KUKA KRL program: DAI_CHECK_GRH_01.src, DAI_CHECK_GRH_01.dat

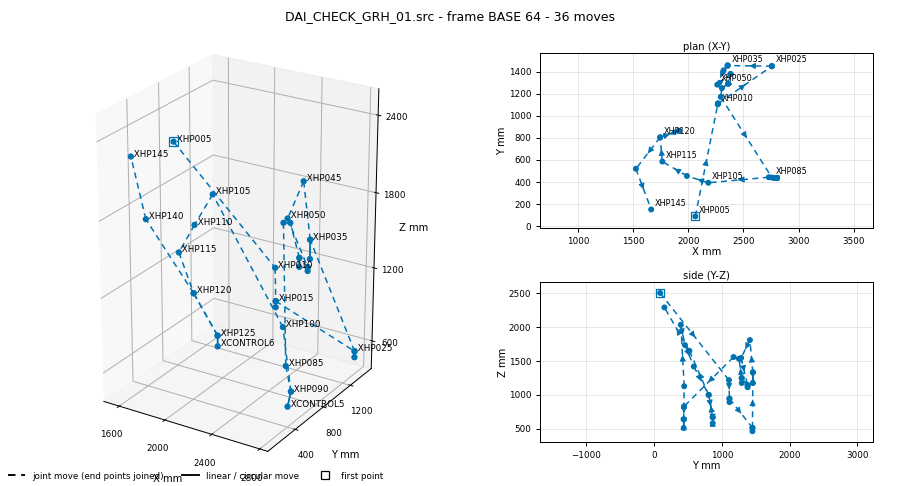
[picture p0: tool path of DAI_CHECK_GRH_01.src in frame BASE 64, 36 of 38 moves have a stored position in this frame; points joined in program order, loops and branches not executed]
--- DAI_CHECK_GRH_01.src ---
&ACCESS RVO
&REL 41
&COMMENT Greiferpruefung
&PARAM TEMPLATE = C:\KRC\roboter\template\vg_appl
&PARAM DISKPATH = KRC:\R1\H_Prog
DEF DAI_CHECK_GRH_01( )
;FOLD INI;%{PE}
  ;FOLD BASISTECH INI
    GLOBAL INTERRUPT DECL 3 WHEN $STOPMESS==TRUE DO IR_STOPM ( )
    INTERRUPT ON 3
    BAS (#INITMOV,0 )
  ;ENDFOLD (BASISTECH INI)
  ;FOLD USER INI
    ;Make your modifications here
  ;ENDFOLD (USER INI)
;ENDFOLD (INI)
;FOLD ; Anlagenbezeichn: HC53_C    Stations-Nr: 060RB_100;%{PE}
;FOLD Parameters ;%{h}
;Params IlfProvider=kukaroboter.basistech.inlineforms.comments.comment; Kuka.Content=Anlagenbezeichn: HC53_C    Stations-Nr: 060RB_100
;ENDFOLD
;ENDFOLD
;FOLD ; Stand / Version: V1.0;%{PE}
;FOLD Parameters ;%{h}
;Params IlfProvider=kukaroboter.basistech.inlineforms.comments.comment; Kuka.Content=Stand / Version: V1.0
;ENDFOLD
;ENDFOLD
;FOLD ; Name Bearbeiter: EBZ-AE;%{PE}
;FOLD Parameters ;%{h}
;Params IlfProvider=kukaroboter.basistech.inlineforms.comments.comment; Kuka.Content=Name Bearbeiter: EBZ-AE
;ENDFOLD
;ENDFOLD
;FOLD ; Translator Version:29.01.2024 - Version 15.08;%{PE}
;FOLD Parameters ;%{h}
;Params IlfProvider=kukaroboter.basistech.inlineforms.comments.comment; Kuka.Content=Translator Version:29.01.2024 - Version 15.08
;ENDFOLD
;ENDFOLD

REPEAT
;FOLD MSG_T1
MSG_SHOW("DAI_H_Prog",#quit,999,"dai_tool_ok_1")
;ENDFOLD

; ***************************************
; A C H T U N G !!! Nur in $T1 abfahren
; ***************************************
UNTIL $T1 == TRUE
;FOLD robot_ok-program
MSG_SHOW("DAI_H_Prog",#quit,999,"dai_rob_ok_0")
DAI_ROBOT_OK ( )
;ENDFOLD

; ***************************************
; Bei Werkzeugwechsel Abfrage ob richtiges Werkzeug angekoppelt ist
; ***************************************
;FOLD MSG_Tool_chg
MSG_BTN("OK")
MSG_SHOW("DAI_H_Prog",#dialog,999,"dai_tool_ok_1",handle,answer)
;ENDFOLD


;FOLD ; This program has been cleaned by KANERT_Makro. High risk of crash!!! Check the program carefully before deleting this comment. ;%{PE}
;FOLD Parameters ;%{h}
;Params IlfProvider=kukaroboter.basistech.inlineforms.comments.comment; Kuka.Content=This program has been cleaned by KANERT_Makro. High risk of crash!!! Check the program carefully before deleting this comment.
;ENDFOLD
WAIT FOR FALSE
;ENDFOLD
;FOLD PTP HOME Vel=100 % DEFAULT;%{PE}
;FOLD Parameters ;%{h}
;Params IlfProvider=kukaroboter.basistech.inlineforms.movement.old; Kuka.IsGlobalPoint=False; Kuka.PointName=HOME; Kuka.BlendingEnabled=False; Kuka.MoveDataPtpName=DEFAULT; Kuka.VelocityPtp=100; Kuka.CurrentCDSetIndex=0; Kuka.MovementParameterFieldEnabled=True; IlfCommand=PTP
;ENDFOLD
$BWDSTART = FALSE
PDAT_ACT = PDEFAULT
FDAT_ACT = FHOME
BAS(#PTP_PARAMS, 100.0)
SET_CD_PARAMS (0)
PTP XHOME
;ENDFOLD

;Dynamische Pruefung Teil vorhanden
;FOLD PartPresent.CheckOff #1:5277, #2:5278, #3:1025, #4:1025, #5:1025, #6:1025, Bounce Time:100, Constant: Yes;%{PE}%
CheckPartPresent(5277,5278,1025,1025,1025,1025,100, True,FALSE)
;ENDFOLD

;Greifer-Ventile betatigen/pruefen
;FOLD DAI_GripValveCheck.Valve2 State:Fixierstift Ausfahren Gs, 060GRH101-QM1;%{PE}%
CheckValveState(2,1)
;ENDFOLD
;FOLD DAI_GripValveCheck.Valve3 State:Spanner Oeffnen Gs, 060GRH101-QM2;%{PE}%
CheckValveState(3,1)
;ENDFOLD
;FOLD DAI_GripValveCheck.Valve4 State:Spanner Oeffnen Gs, 060GRH101-QM3;%{PE}%
CheckValveState(4,1)
;ENDFOLD

;FOLD PTP HP005 Vel=100 % PDAT1 Tool[64]:Zero Base[64]:Zero;%{PE}
;FOLD Parameters ;%{h}
;Params IlfProvider=kukaroboter.basistech.inlineforms.movement.old; Kuka.IsGlobalPoint=False; Kuka.PointName=HP005; Kuka.BlendingEnabled=False; Kuka.MoveDataPtpName=PDAT1; Kuka.VelocityPtp=100; Kuka.CurrentCDSetIndex=0; Kuka.MovementParameterFieldEnabled=True; IlfCommand=PTP
;ENDFOLD
$BWDSTART = FALSE
PDAT_ACT = PPDAT1
FDAT_ACT = FHP005
BAS(#PTP_PARAMS, 100.0)
SET_CD_PARAMS (0)
PTP XHP005
;ENDFOLD
;FOLD PTP HP010 Vel=100 % PDAT2 Tool[64]:Zero Base[64]:Zero;%{PE}
;FOLD Parameters ;%{h}
;Params IlfProvider=kukaroboter.basistech.inlineforms.movement.old; Kuka.IsGlobalPoint=False; Kuka.PointName=HP010; Kuka.BlendingEnabled=False; Kuka.MoveDataPtpName=PDAT2; Kuka.VelocityPtp=100; Kuka.CurrentCDSetIndex=0; Kuka.MovementParameterFieldEnabled=True; IlfCommand=PTP
;ENDFOLD
$BWDSTART = FALSE
PDAT_ACT = PPDAT2
FDAT_ACT = FHP010
BAS(#PTP_PARAMS, 100.0)
SET_CD_PARAMS (0)
PTP XHP010
;ENDFOLD
;FOLD PTP HP015 Vel=100 % PDAT3 Tool[64]:Zero Base[64]:Zero;%{PE}
;FOLD Parameters ;%{h}
;Params IlfProvider=kukaroboter.basistech.inlineforms.movement.old; Kuka.IsGlobalPoint=False; Kuka.PointName=HP015; Kuka.BlendingEnabled=False; Kuka.MoveDataPtpName=PDAT3; Kuka.VelocityPtp=100; Kuka.CurrentCDSetIndex=0; Kuka.MovementParameterFieldEnabled=True; IlfCommand=PTP
;ENDFOLD
$BWDSTART = FALSE
PDAT_ACT = PPDAT3
FDAT_ACT = FHP015
BAS(#PTP_PARAMS, 100.0)
SET_CD_PARAMS (0)
PTP XHP015
;ENDFOLD

; ***************************************
; Stift ausfahren
; ***************************************

; ***************************************
;FOLD Kontrollspitzen anbringen
MSG_BTN("OK")
MSG_SHOW("DAI_H_PROG",#dialog,999,"dai_tool_ok_7",handle,answer)
;ENDFOLD
;FOLD WAIT FOR ( IN 1026 'Vordefinierte Eingang immer ruckgesetzt.' )  ;%{PE}
;FOLD Parameters ;%{h}
;Params IlfProvider=kukaroboter.basistech.inlineforms.logics.waitfor; Kuka.WaitLogicTerm1=None; Kuka.WaitForNot1=False; Kuka.WaitLogicOp2.Term1=None; Kuka.WaitForNot2.Term1=False; Kuka.WaitForSysVar2.Term1=IN; Kuka.WaitForIndex2.Term1=1026; Kuka.WaitForIndexName2.Term1=Vordefinierte Eingang immer ruckgesetzt.; Kuka.WaitForTermNumbers=1; Kuka.WaitForOpNumbers=2; Kuka.WaitForCont=False
;ENDFOLD
WAIT FOR  ( $IN[1026] )
;ENDFOLD

; ***************************************
;FOLD ;Kontrollposition 1 QMXMMYY mit Tool 64 ;%{PE}
;FOLD Parameters ;%{h}
;Params IlfProvider=kukaroboter.basistech.inlineforms.comments.comment; Kuka.Content=Kontrollposition 1 QMXMMYY mit Tool 64
;ENDFOLD
;ENDFOLD
;FOLD LIN CONTROL1 Vel=0.2 m/s CPDAT4 Tool[64]:Zero Base[64]:Zero ;%{PE}
;FOLD Parameters ;%{h}
;Params IlfProvider=kukaroboter.basistech.inlineforms.movement.old; Kuka.IsGlobalPoint=False; Kuka.PointName=CONTROL1; Kuka.BlendingEnabled=False; Kuka.MoveDataName=CPDAT4; Kuka.VelocityPath=0.2; Kuka.CurrentCDSetIndex=0; Kuka.MovementParameterFieldEnabled=True; IlfCommand=LIN
;ENDFOLD
$BWDSTART = FALSE
LDAT_ACT = LCPDAT4
FDAT_ACT = FCONTROL1
BAS(#CP_PARAMS, 0.2)
SET_CD_PARAMS (0)
LIN XCONTROL1
;ENDFOLD

;FOLD WAIT FOR ( IN 1026 'Vordefinierte Eingang immer ruckgesetzt.' )  ;%{PE}
;FOLD Parameters ;%{h}
;Params IlfProvider=kukaroboter.basistech.inlineforms.logics.waitfor; Kuka.WaitLogicTerm1=None; Kuka.WaitForNot1=False; Kuka.WaitLogicOp2.Term1=None; Kuka.WaitForNot2.Term1=False; Kuka.WaitForSysVar2.Term1=IN; Kuka.WaitForIndex2.Term1=1026; Kuka.WaitForIndexName2.Term1=Vordefinierte Eingang immer ruckgesetzt.; Kuka.WaitForTermNumbers=1; Kuka.WaitForOpNumbers=2; Kuka.WaitForCont=False
;ENDFOLD
WAIT FOR  ( $IN[1026] )
;ENDFOLD

;FOLD LIN HP020 Vel=0.2 m/s CPDAT5 Tool[64]:Zero Base[64]:Zero ;%{PE}
;FOLD Parameters ;%{h}
;Params IlfProvider=kukaroboter.basistech.inlineforms.movement.old; Kuka.IsGlobalPoint=False; Kuka.PointName=HP020; Kuka.BlendingEnabled=False; Kuka.MoveDataName=CPDAT5; Kuka.VelocityPath=0.2; Kuka.CurrentCDSetIndex=0; Kuka.MovementParameterFieldEnabled=True; IlfCommand=LIN
;ENDFOLD
$BWDSTART = FALSE
LDAT_ACT = LCPDAT5
FDAT_ACT = FHP020
BAS(#CP_PARAMS, 0.2)
SET_CD_PARAMS (0)
LIN XHP020
;ENDFOLD

; ***************************************
; Die naechsten 3 Punkte werden mit Tool[10] angefahren
; ***************************************
;FOLD PTP HP025 Vel=100 % PDAT6 Tool[10]:GRH_01_ZBHC_O Base[64]:Zero;%{PE}
;FOLD Parameters ;%{h}
;Params IlfProvider=kukaroboter.basistech.inlineforms.movement.old; Kuka.IsGlobalPoint=False; Kuka.PointName=HP025; Kuka.BlendingEnabled=False; Kuka.MoveDataPtpName=PDAT6; Kuka.VelocityPtp=100; Kuka.CurrentCDSetIndex=0; Kuka.MovementParameterFieldEnabled=True; IlfCommand=PTP
;ENDFOLD
$BWDSTART = FALSE
PDAT_ACT = PPDAT6
FDAT_ACT = FHP025
BAS(#PTP_PARAMS, 100.0)
SET_CD_PARAMS (0)
PTP XHP025
;ENDFOLD

;FOLD ; Kontrollposition 1A QM1MM01 mit Tool 10 ;%{PE}
;FOLD Parameters ;%{h}
;Params IlfProvider=kukaroboter.basistech.inlineforms.comments.comment; Kuka.Content=Kontrollposition 1A QM1MM01 mit Tool 10
;ENDFOLD
;ENDFOLD
;FOLD LIN CONTROL1A Vel=0.2 m/s CPDAT7 Tool[10]:GRH_01_ZBHC_O Base[64]:Zero ;%{PE}
;FOLD Parameters ;%{h}
;Params IlfProvider=kukaroboter.basistech.inlineforms.movement.old; Kuka.IsGlobalPoint=False; Kuka.PointName=CONTROL1A; Kuka.BlendingEnabled=False; Kuka.MoveDataName=CPDAT7; Kuka.VelocityPath=0.2; Kuka.CurrentCDSetIndex=0; Kuka.MovementParameterFieldEnabled=True; IlfCommand=LIN
;ENDFOLD
$BWDSTART = FALSE
LDAT_ACT = LCPDAT7
FDAT_ACT = FCONTROL1A
BAS(#CP_PARAMS, 0.2)
SET_CD_PARAMS (0)
LIN XCONTROL1A
;ENDFOLD

;FOLD WAIT FOR ( IN 1026 'Vordefinierte Eingang immer ruckgesetzt.' )  ;%{PE}
;FOLD Parameters ;%{h}
;Params IlfProvider=kukaroboter.basistech.inlineforms.logics.waitfor; Kuka.WaitLogicTerm1=None; Kuka.WaitForNot1=False; Kuka.WaitLogicOp2.Term1=None; Kuka.WaitForNot2.Term1=False; Kuka.WaitForSysVar2.Term1=IN; Kuka.WaitForIndex2.Term1=1026; Kuka.WaitForIndexName2.Term1=Vordefinierte Eingang immer ruckgesetzt.; Kuka.WaitForTermNumbers=1; Kuka.WaitForOpNumbers=2; Kuka.WaitForCont=False
;ENDFOLD
WAIT FOR  ( $IN[1026] )
;ENDFOLD

;FOLD LIN HP030 Vel=0.2 m/s CPDAT8 Tool[10]:GRH_01_ZBHC_O Base[64]:Zero ;%{PE}
;FOLD Parameters ;%{h}
;Params IlfProvider=kukaroboter.basistech.inlineforms.movement.old; Kuka.IsGlobalPoint=False; Kuka.PointName=HP030; Kuka.BlendingEnabled=False; Kuka.MoveDataName=CPDAT8; Kuka.VelocityPath=0.2; Kuka.CurrentCDSetIndex=0; Kuka.MovementParameterFieldEnabled=True; IlfCommand=LIN
;ENDFOLD
$BWDSTART = FALSE
LDAT_ACT = LCPDAT8
FDAT_ACT = FHP030
BAS(#CP_PARAMS, 0.2)
SET_CD_PARAMS (0)
LIN XHP030
;ENDFOLD
;FOLD PTP HP035 Vel=100 % PDAT9 Tool[64]:Zero Base[64]:Zero;%{PE}
;FOLD Parameters ;%{h}
;Params IlfProvider=kukaroboter.basistech.inlineforms.movement.old; Kuka.IsGlobalPoint=False; Kuka.PointName=HP035; Kuka.BlendingEnabled=False; Kuka.MoveDataPtpName=PDAT9; Kuka.VelocityPtp=100; Kuka.CurrentCDSetIndex=0; Kuka.MovementParameterFieldEnabled=True; IlfCommand=PTP
;ENDFOLD
$BWDSTART = FALSE
PDAT_ACT = PPDAT9
FDAT_ACT = FHP035
BAS(#PTP_PARAMS, 100.0)
SET_CD_PARAMS (0)
PTP XHP035
;ENDFOLD

;FOLD ; Kontrollposition 2 QM2MM1 mit Tool 64 ;%{PE}
;FOLD Parameters ;%{h}
;Params IlfProvider=kukaroboter.basistech.inlineforms.comments.comment; Kuka.Content=Kontrollposition 2 QM2MM1 mit Tool 64
;ENDFOLD
;ENDFOLD
;FOLD LIN CONTROL2 Vel=0.2 m/s CPDAT10 Tool[64]:Zero Base[64]:Zero ;%{PE}
;FOLD Parameters ;%{h}
;Params IlfProvider=kukaroboter.basistech.inlineforms.movement.old; Kuka.IsGlobalPoint=False; Kuka.PointName=CONTROL2; Kuka.BlendingEnabled=False; Kuka.MoveDataName=CPDAT10; Kuka.VelocityPath=0.2; Kuka.CurrentCDSetIndex=0; Kuka.MovementParameterFieldEnabled=True; IlfCommand=LIN
;ENDFOLD
$BWDSTART = FALSE
LDAT_ACT = LCPDAT10
FDAT_ACT = FCONTROL2
BAS(#CP_PARAMS, 0.2)
SET_CD_PARAMS (0)
LIN XCONTROL2
;ENDFOLD

;FOLD WAIT FOR ( IN 1026 'Vordefinierte Eingang immer ruckgesetzt.' )  ;%{PE}
;FOLD Parameters ;%{h}
;Params IlfProvider=kukaroboter.basistech.inlineforms.logics.waitfor; Kuka.WaitLogicTerm1=None; Kuka.WaitForNot1=False; Kuka.WaitLogicOp2.Term1=None; Kuka.WaitForNot2.Term1=False; Kuka.WaitForSysVar2.Term1=IN; Kuka.WaitForIndex2.Term1=1026; Kuka.WaitForIndexName2.Term1=Vordefinierte Eingang immer ruckgesetzt.; Kuka.WaitForTermNumbers=1; Kuka.WaitForOpNumbers=2; Kuka.WaitForCont=False
;ENDFOLD
WAIT FOR  ( $IN[1026] )
;ENDFOLD

;FOLD LIN HP040 Vel=0.2 m/s CPDAT11 Tool[64]:Zero Base[64]:Zero ;%{PE}
;FOLD Parameters ;%{h}
;Params IlfProvider=kukaroboter.basistech.inlineforms.movement.old; Kuka.IsGlobalPoint=False; Kuka.PointName=HP040; Kuka.BlendingEnabled=False; Kuka.MoveDataName=CPDAT11; Kuka.VelocityPath=0.2; Kuka.CurrentCDSetIndex=0; Kuka.MovementParameterFieldEnabled=True; IlfCommand=LIN
;ENDFOLD
$BWDSTART = FALSE
LDAT_ACT = LCPDAT11
FDAT_ACT = FHP040
BAS(#CP_PARAMS, 0.2)
SET_CD_PARAMS (0)
LIN XHP040
;ENDFOLD
;FOLD PTP HP045 Vel=100 % PDAT12 Tool[64]:Zero Base[64]:Zero;%{PE}
;FOLD Parameters ;%{h}
;Params IlfProvider=kukaroboter.basistech.inlineforms.movement.old; Kuka.IsGlobalPoint=False; Kuka.PointName=HP045; Kuka.BlendingEnabled=False; Kuka.MoveDataPtpName=PDAT12; Kuka.VelocityPtp=100; Kuka.CurrentCDSetIndex=0; Kuka.MovementParameterFieldEnabled=True; IlfCommand=PTP
;ENDFOLD
$BWDSTART = FALSE
PDAT_ACT = PPDAT12
FDAT_ACT = FHP045
BAS(#PTP_PARAMS, 100.0)
SET_CD_PARAMS (0)
PTP XHP045
;ENDFOLD
;FOLD PTP HP050 Vel=100 % PDAT13 Tool[64]:Zero Base[64]:Zero;%{PE}
;FOLD Parameters ;%{h}
;Params IlfProvider=kukaroboter.basistech.inlineforms.movement.old; Kuka.IsGlobalPoint=False; Kuka.PointName=HP050; Kuka.BlendingEnabled=False; Kuka.MoveDataPtpName=PDAT13; Kuka.VelocityPtp=100; Kuka.CurrentCDSetIndex=0; Kuka.MovementParameterFieldEnabled=True; IlfCommand=PTP
;ENDFOLD
$BWDSTART = FALSE
PDAT_ACT = PPDAT13
FDAT_ACT = FHP050
BAS(#PTP_PARAMS, 100.0)
SET_CD_PARAMS (0)
PTP XHP050
;ENDFOLD
;FOLD PTP HP055 Vel=100 % PDAT14 Tool[64]:Zero Base[64]:Zero;%{PE}
;FOLD Parameters ;%{h}
;Params IlfProvider=kukaroboter.basistech.inlineforms.movement.old; Kuka.IsGlobalPoint=False; Kuka.PointName=HP055; Kuka.BlendingEnabled=False; Kuka.MoveDataPtpName=PDAT14; Kuka.VelocityPtp=100; Kuka.CurrentCDSetIndex=0; Kuka.MovementParameterFieldEnabled=True; IlfCommand=PTP
;ENDFOLD
$BWDSTART = FALSE
PDAT_ACT = PPDAT14
FDAT_ACT = FHP055
BAS(#PTP_PARAMS, 100.0)
SET_CD_PARAMS (0)
PTP XHP055
;ENDFOLD

;FOLD ; Kontrollposition 3 QM1MM01 mit Tool 64 ;%{PE}
;FOLD Parameters ;%{h}
;Params IlfProvider=kukaroboter.basistech.inlineforms.comments.comment; Kuka.Content=Kontrollposition 3 QM1MM01 mit Tool 64
;ENDFOLD
;ENDFOLD
;FOLD LIN CONTROL3 Vel=0.2 m/s CPDAT15 Tool[64]:Zero Base[64]:Zero ;%{PE}
;FOLD Parameters ;%{h}
;Params IlfProvider=kukaroboter.basistech.inlineforms.movement.old; Kuka.IsGlobalPoint=False; Kuka.PointName=CONTROL3; Kuka.BlendingEnabled=False; Kuka.MoveDataName=CPDAT15; Kuka.VelocityPath=0.2; Kuka.CurrentCDSetIndex=0; Kuka.MovementParameterFieldEnabled=True; IlfCommand=LIN
;ENDFOLD
$BWDSTART = FALSE
LDAT_ACT = LCPDAT15
FDAT_ACT = FCONTROL3
BAS(#CP_PARAMS, 0.2)
SET_CD_PARAMS (0)
LIN XCONTROL3
;ENDFOLD

;FOLD WAIT FOR ( IN 1026 'Vordefinierte Eingang immer ruckgesetzt.' )  ;%{PE}
;FOLD Parameters ;%{h}
;Params IlfProvider=kukaroboter.basistech.inlineforms.logics.waitfor; Kuka.WaitLogicTerm1=None; Kuka.WaitForNot1=False; Kuka.WaitLogicOp2.Term1=None; Kuka.WaitForNot2.Term1=False; Kuka.WaitForSysVar2.Term1=IN; Kuka.WaitForIndex2.Term1=1026; Kuka.WaitForIndexName2.Term1=Vordefinierte Eingang immer ruckgesetzt.; Kuka.WaitForTermNumbers=1; Kuka.WaitForOpNumbers=2; Kuka.WaitForCont=False
;ENDFOLD
WAIT FOR  ( $IN[1026] )
;ENDFOLD

;FOLD LIN HP060 Vel=0.2 m/s CPDAT16 Tool[64]:Zero Base[64]:Zero ;%{PE}
;FOLD Parameters ;%{h}
;Params IlfProvider=kukaroboter.basistech.inlineforms.movement.old; Kuka.IsGlobalPoint=False; Kuka.PointName=HP060; Kuka.BlendingEnabled=False; Kuka.MoveDataName=CPDAT16; Kuka.VelocityPath=0.2; Kuka.CurrentCDSetIndex=0; Kuka.MovementParameterFieldEnabled=True; IlfCommand=LIN
;ENDFOLD
$BWDSTART = FALSE
LDAT_ACT = LCPDAT16
FDAT_ACT = FHP060
BAS(#CP_PARAMS, 0.2)
SET_CD_PARAMS (0)
LIN XHP060
;ENDFOLD
;FOLD PTP HP065 Vel=100 % PDAT17 Tool[64]:Zero Base[64]:Zero;%{PE}
;FOLD Parameters ;%{h}
;Params IlfProvider=kukaroboter.basistech.inlineforms.movement.old; Kuka.IsGlobalPoint=False; Kuka.PointName=HP065; Kuka.BlendingEnabled=False; Kuka.MoveDataPtpName=PDAT17; Kuka.VelocityPtp=100; Kuka.CurrentCDSetIndex=0; Kuka.MovementParameterFieldEnabled=True; IlfCommand=PTP
;ENDFOLD
$BWDSTART = FALSE
PDAT_ACT = PPDAT17
FDAT_ACT = FHP065
BAS(#PTP_PARAMS, 100.0)
SET_CD_PARAMS (0)
PTP XHP065
;ENDFOLD

;FOLD ; Kontrollposition 4 QM3MM1 mit Tool 64 ;%{PE}
;FOLD Parameters ;%{h}
;Params IlfProvider=kukaroboter.basistech.inlineforms.comments.comment; Kuka.Content=Kontrollposition 4 QM3MM1 mit Tool 64
;ENDFOLD
;ENDFOLD
;FOLD LIN CONTROL4 Vel=0.2 m/s CPDAT18 Tool[64]:Zero Base[64]:Zero ;%{PE}
;FOLD Parameters ;%{h}
;Params IlfProvider=kukaroboter.basistech.inlineforms.movement.old; Kuka.IsGlobalPoint=False; Kuka.PointName=CONTROL4; Kuka.BlendingEnabled=False; Kuka.MoveDataName=CPDAT18; Kuka.VelocityPath=0.2; Kuka.CurrentCDSetIndex=0; Kuka.MovementParameterFieldEnabled=True; IlfCommand=LIN
;ENDFOLD
$BWDSTART = FALSE
LDAT_ACT = LCPDAT18
FDAT_ACT = FCONTROL4
BAS(#CP_PARAMS, 0.2)
SET_CD_PARAMS (0)
LIN XCONTROL4
;ENDFOLD

;FOLD WAIT FOR ( IN 1026 'Vordefinierte Eingang immer ruckgesetzt.' )  ;%{PE}
;FOLD Parameters ;%{h}
;Params IlfProvider=kukaroboter.basistech.inlineforms.logics.waitfor; Kuka.WaitLogicTerm1=None; Kuka.WaitForNot1=False; Kuka.WaitLogicOp2.Term1=None; Kuka.WaitForNot2.Term1=False; Kuka.WaitForSysVar2.Term1=IN; Kuka.WaitForIndex2.Term1=1026; Kuka.WaitForIndexName2.Term1=Vordefinierte Eingang immer ruckgesetzt.; Kuka.WaitForTermNumbers=1; Kuka.WaitForOpNumbers=2; Kuka.WaitForCont=False
;ENDFOLD
WAIT FOR  ( $IN[1026] )
;ENDFOLD

;FOLD LIN HP070 Vel=0.2 m/s CPDAT19 Tool[64]:Zero Base[64]:Zero ;%{PE}
;FOLD Parameters ;%{h}
;Params IlfProvider=kukaroboter.basistech.inlineforms.movement.old; Kuka.IsGlobalPoint=False; Kuka.PointName=HP070; Kuka.BlendingEnabled=False; Kuka.MoveDataName=CPDAT19; Kuka.VelocityPath=0.2; Kuka.CurrentCDSetIndex=0; Kuka.MovementParameterFieldEnabled=True; IlfCommand=LIN
;ENDFOLD
$BWDSTART = FALSE
LDAT_ACT = LCPDAT19
FDAT_ACT = FHP070
BAS(#CP_PARAMS, 0.2)
SET_CD_PARAMS (0)
LIN XHP070
;ENDFOLD
;FOLD PTP HP075 Vel=100 % PDAT20 Tool[64]:Zero Base[64]:Zero;%{PE}
;FOLD Parameters ;%{h}
;Params IlfProvider=kukaroboter.basistech.inlineforms.movement.old; Kuka.IsGlobalPoint=False; Kuka.PointName=HP075; Kuka.BlendingEnabled=False; Kuka.MoveDataPtpName=PDAT20; Kuka.VelocityPtp=100; Kuka.CurrentCDSetIndex=0; Kuka.MovementParameterFieldEnabled=True; IlfCommand=PTP
;ENDFOLD
$BWDSTART = FALSE
PDAT_ACT = PPDAT20
FDAT_ACT = FHP075
BAS(#PTP_PARAMS, 100.0)
SET_CD_PARAMS (0)
PTP XHP075
;ENDFOLD
;FOLD PTP HP080 Vel=100 % PDAT21 Tool[64]:Zero Base[64]:Zero;%{PE}
;FOLD Parameters ;%{h}
;Params IlfProvider=kukaroboter.basistech.inlineforms.movement.old; Kuka.IsGlobalPoint=False; Kuka.PointName=HP080; Kuka.BlendingEnabled=False; Kuka.MoveDataPtpName=PDAT21; Kuka.VelocityPtp=100; Kuka.CurrentCDSetIndex=0; Kuka.MovementParameterFieldEnabled=True; IlfCommand=PTP
;ENDFOLD
$BWDSTART = FALSE
PDAT_ACT = PPDAT21
FDAT_ACT = FHP080
BAS(#PTP_PARAMS, 100.0)
SET_CD_PARAMS (0)
PTP XHP080
;ENDFOLD
;FOLD PTP HP085 Vel=100 % PDAT22 Tool[64]:Zero Base[64]:Zero;%{PE}
;FOLD Parameters ;%{h}
;Params IlfProvider=kukaroboter.basistech.inlineforms.movement.old; Kuka.IsGlobalPoint=False; Kuka.PointName=HP085; Kuka.BlendingEnabled=False; Kuka.MoveDataPtpName=PDAT22; Kuka.VelocityPtp=100; Kuka.CurrentCDSetIndex=0; Kuka.MovementParameterFieldEnabled=True; IlfCommand=PTP
;ENDFOLD
$BWDSTART = FALSE
PDAT_ACT = PPDAT22
FDAT_ACT = FHP085
BAS(#PTP_PARAMS, 100.0)
SET_CD_PARAMS (0)
PTP XHP085
;ENDFOLD
;FOLD PTP HP090 Vel=100 % PDAT23 Tool[64]:Zero Base[64]:Zero;%{PE}
;FOLD Parameters ;%{h}
;Params IlfProvider=kukaroboter.basistech.inlineforms.movement.old; Kuka.IsGlobalPoint=False; Kuka.PointName=HP090; Kuka.BlendingEnabled=False; Kuka.MoveDataPtpName=PDAT23; Kuka.VelocityPtp=100; Kuka.CurrentCDSetIndex=0; Kuka.MovementParameterFieldEnabled=True; IlfCommand=PTP
;ENDFOLD
$BWDSTART = FALSE
PDAT_ACT = PPDAT23
FDAT_ACT = FHP090
BAS(#PTP_PARAMS, 100.0)
SET_CD_PARAMS (0)
PTP XHP090
;ENDFOLD

;FOLD ; Kontrollposition 5 QM3MM2 mit Tool 64 ;%{PE}
;FOLD Parameters ;%{h}
;Params IlfProvider=kukaroboter.basistech.inlineforms.comments.comment; Kuka.Content=Kontrollposition 5 QM3MM2 mit Tool 64
;ENDFOLD
;ENDFOLD
;FOLD LIN CONTROL5 Vel=0.2 m/s CPDAT24 Tool[64]:Zero Base[64]:Zero ;%{PE}
;FOLD Parameters ;%{h}
;Params IlfProvider=kukaroboter.basistech.inlineforms.movement.old; Kuka.IsGlobalPoint=False; Kuka.PointName=CONTROL5; Kuka.BlendingEnabled=False; Kuka.MoveDataName=CPDAT24; Kuka.VelocityPath=0.2; Kuka.CurrentCDSetIndex=0; Kuka.MovementParameterFieldEnabled=True; IlfCommand=LIN
;ENDFOLD
$BWDSTART = FALSE
LDAT_ACT = LCPDAT24
FDAT_ACT = FCONTROL5
BAS(#CP_PARAMS, 0.2)
SET_CD_PARAMS (0)
LIN XCONTROL5
;ENDFOLD

;FOLD WAIT FOR ( IN 1026 'Vordefinierte Eingang immer ruckgesetzt.' )  ;%{PE}
;FOLD Parameters ;%{h}
;Params IlfProvider=kukaroboter.basistech.inlineforms.logics.waitfor; Kuka.WaitLogicTerm1=None; Kuka.WaitForNot1=False; Kuka.WaitLogicOp2.Term1=None; Kuka.WaitForNot2.Term1=False; Kuka.WaitForSysVar2.Term1=IN; Kuka.WaitForIndex2.Term1=1026; Kuka.WaitForIndexName2.Term1=Vordefinierte Eingang immer ruckgesetzt.; Kuka.WaitForTermNumbers=1; Kuka.WaitForOpNumbers=2; Kuka.WaitForCont=False
;ENDFOLD
WAIT FOR  ( $IN[1026] )
;ENDFOLD

;FOLD LIN HP095 Vel=0.2 m/s CPDAT25 Tool[64]:Zero Base[64]:Zero ;%{PE}
;FOLD Parameters ;%{h}
;Params IlfProvider=kukaroboter.basistech.inlineforms.movement.old; Kuka.IsGlobalPoint=False; Kuka.PointName=HP095; Kuka.BlendingEnabled=False; Kuka.MoveDataName=CPDAT25; Kuka.VelocityPath=0.2; Kuka.CurrentCDSetIndex=0; Kuka.MovementParameterFieldEnabled=True; IlfCommand=LIN
;ENDFOLD
$BWDSTART = FALSE
LDAT_ACT = LCPDAT25
FDAT_ACT = FHP095
BAS(#CP_PARAMS, 0.2)
SET_CD_PARAMS (0)
LIN XHP095
;ENDFOLD
;FOLD PTP HP100 Vel=100 % PDAT26 Tool[64]:Zero Base[64]:Zero;%{PE}
;FOLD Parameters ;%{h}
;Params IlfProvider=kukaroboter.basistech.inlineforms.movement.old; Kuka.IsGlobalPoint=False; Kuka.PointName=HP100; Kuka.BlendingEnabled=False; Kuka.MoveDataPtpName=PDAT26; Kuka.VelocityPtp=100; Kuka.CurrentCDSetIndex=0; Kuka.MovementParameterFieldEnabled=True; IlfCommand=PTP
;ENDFOLD
$BWDSTART = FALSE
PDAT_ACT = PPDAT26
FDAT_ACT = FHP100
BAS(#PTP_PARAMS, 100.0)
SET_CD_PARAMS (0)
PTP XHP100
;ENDFOLD
;FOLD PTP HP105 Vel=100 % PDAT27 Tool[64]:Zero Base[64]:Zero;%{PE}
;FOLD Parameters ;%{h}
;Params IlfProvider=kukaroboter.basistech.inlineforms.movement.old; Kuka.IsGlobalPoint=False; Kuka.PointName=HP105; Kuka.BlendingEnabled=False; Kuka.MoveDataPtpName=PDAT27; Kuka.VelocityPtp=100; Kuka.CurrentCDSetIndex=0; Kuka.MovementParameterFieldEnabled=True; IlfCommand=PTP
;ENDFOLD
$BWDSTART = FALSE
PDAT_ACT = PPDAT27
FDAT_ACT = FHP105
BAS(#PTP_PARAMS, 100.0)
SET_CD_PARAMS (0)
PTP XHP105
;ENDFOLD
;FOLD PTP HP110 Vel=100 % PDAT28 Tool[64]:Zero Base[64]:Zero;%{PE}
;FOLD Parameters ;%{h}
;Params IlfProvider=kukaroboter.basistech.inlineforms.movement.old; Kuka.IsGlobalPoint=False; Kuka.PointName=HP110; Kuka.BlendingEnabled=False; Kuka.MoveDataPtpName=PDAT28; Kuka.VelocityPtp=100; Kuka.CurrentCDSetIndex=0; Kuka.MovementParameterFieldEnabled=True; IlfCommand=PTP
;ENDFOLD
$BWDSTART = FALSE
PDAT_ACT = PPDAT28
FDAT_ACT = FHP110
BAS(#PTP_PARAMS, 100.0)
SET_CD_PARAMS (0)
PTP XHP110
;ENDFOLD
;FOLD PTP HP115 Vel=100 % PDAT29 Tool[64]:Zero Base[64]:Zero;%{PE}
;FOLD Parameters ;%{h}
;Params IlfProvider=kukaroboter.basistech.inlineforms.movement.old; Kuka.IsGlobalPoint=False; Kuka.PointName=HP115; Kuka.BlendingEnabled=False; Kuka.MoveDataPtpName=PDAT29; Kuka.VelocityPtp=100; Kuka.CurrentCDSetIndex=0; Kuka.MovementParameterFieldEnabled=True; IlfCommand=PTP
;ENDFOLD
$BWDSTART = FALSE
PDAT_ACT = PPDAT29
FDAT_ACT = FHP115
BAS(#PTP_PARAMS, 100.0)
SET_CD_PARAMS (0)
PTP XHP115
;ENDFOLD
;FOLD PTP HP120 Vel=100 % PDAT30 Tool[64]:Zero Base[64]:Zero;%{PE}
;FOLD Parameters ;%{h}
;Params IlfProvider=kukaroboter.basistech.inlineforms.movement.old; Kuka.IsGlobalPoint=False; Kuka.PointName=HP120; Kuka.BlendingEnabled=False; Kuka.MoveDataPtpName=PDAT30; Kuka.VelocityPtp=100; Kuka.CurrentCDSetIndex=0; Kuka.MovementParameterFieldEnabled=True; IlfCommand=PTP
;ENDFOLD
$BWDSTART = FALSE
PDAT_ACT = PPDAT30
FDAT_ACT = FHP120
BAS(#PTP_PARAMS, 100.0)
SET_CD_PARAMS (0)
PTP XHP120
;ENDFOLD
;FOLD PTP HP125 Vel=100 % PDAT31 Tool[64]:Zero Base[64]:Zero;%{PE}
;FOLD Parameters ;%{h}
;Params IlfProvider=kukaroboter.basistech.inlineforms.movement.old; Kuka.IsGlobalPoint=False; Kuka.PointName=HP125; Kuka.BlendingEnabled=False; Kuka.MoveDataPtpName=PDAT31; Kuka.VelocityPtp=100; Kuka.CurrentCDSetIndex=0; Kuka.MovementParameterFieldEnabled=True; IlfCommand=PTP
;ENDFOLD
$BWDSTART = FALSE
PDAT_ACT = PPDAT31
FDAT_ACT = FHP125
BAS(#PTP_PARAMS, 100.0)
SET_CD_PARAMS (0)
PTP XHP125
;ENDFOLD

;FOLD ; Kontrollposition 6 QM2MM2 mit Tool 64 ;%{PE}
;FOLD Parameters ;%{h}
;Params IlfProvider=kukaroboter.basistech.inlineforms.comments.comment; Kuka.Content=Kontrollposition 6 QM2MM2 mit Tool 64
;ENDFOLD
;ENDFOLD
;FOLD LIN CONTROL6 Vel=0.2 m/s CPDAT32 Tool[64]:Zero Base[64]:Zero ;%{PE}
;FOLD Parameters ;%{h}
;Params IlfProvider=kukaroboter.basistech.inlineforms.movement.old; Kuka.IsGlobalPoint=False; Kuka.PointName=CONTROL6; Kuka.BlendingEnabled=False; Kuka.MoveDataName=CPDAT32; Kuka.VelocityPath=0.2; Kuka.CurrentCDSetIndex=0; Kuka.MovementParameterFieldEnabled=True; IlfCommand=LIN
;ENDFOLD
$BWDSTART = FALSE
LDAT_ACT = LCPDAT32
FDAT_ACT = FCONTROL6
BAS(#CP_PARAMS, 0.2)
SET_CD_PARAMS (0)
LIN XCONTROL6
;ENDFOLD

;FOLD WAIT FOR ( IN 1026 'Vordefinierte Eingang immer ruckgesetzt.' )  ;%{PE}
;FOLD Parameters ;%{h}
;Params IlfProvider=kukaroboter.basistech.inlineforms.logics.waitfor; Kuka.WaitLogicTerm1=None; Kuka.WaitForNot1=False; Kuka.WaitLogicOp2.Term1=None; Kuka.WaitForNot2.Term1=False; Kuka.WaitForSysVar2.Term1=IN; Kuka.WaitForIndex2.Term1=1026; Kuka.WaitForIndexName2.Term1=Vordefinierte Eingang immer ruckgesetzt.; Kuka.WaitForTermNumbers=1; Kuka.WaitForOpNumbers=2; Kuka.WaitForCont=False
;ENDFOLD
WAIT FOR  ( $IN[1026] )
;ENDFOLD

;FOLD LIN HP130 Vel=0.2 m/s CPDAT33 Tool[64]:Zero Base[64]:Zero ;%{PE}
;FOLD Parameters ;%{h}
;Params IlfProvider=kukaroboter.basistech.inlineforms.movement.old; Kuka.IsGlobalPoint=False; Kuka.PointName=HP130; Kuka.BlendingEnabled=False; Kuka.MoveDataName=CPDAT33; Kuka.VelocityPath=0.2; Kuka.CurrentCDSetIndex=0; Kuka.MovementParameterFieldEnabled=True; IlfCommand=LIN
;ENDFOLD
$BWDSTART = FALSE
LDAT_ACT = LCPDAT33
FDAT_ACT = FHP130
BAS(#CP_PARAMS, 0.2)
SET_CD_PARAMS (0)
LIN XHP130
;ENDFOLD
;FOLD PTP HP135 Vel=100 % PDAT34 Tool[64]:Zero Base[64]:Zero;%{PE}
;FOLD Parameters ;%{h}
;Params IlfProvider=kukaroboter.basistech.inlineforms.movement.old; Kuka.IsGlobalPoint=False; Kuka.PointName=HP135; Kuka.BlendingEnabled=False; Kuka.MoveDataPtpName=PDAT34; Kuka.VelocityPtp=100; Kuka.CurrentCDSetIndex=0; Kuka.MovementParameterFieldEnabled=True; IlfCommand=PTP
;ENDFOLD
$BWDSTART = FALSE
PDAT_ACT = PPDAT34
FDAT_ACT = FHP135
BAS(#PTP_PARAMS, 100.0)
SET_CD_PARAMS (0)
PTP XHP135
;ENDFOLD
;FOLD PTP HP140 Vel=100 % PDAT35 Tool[64]:Zero Base[64]:Zero;%{PE}
;FOLD Parameters ;%{h}
;Params IlfProvider=kukaroboter.basistech.inlineforms.movement.old; Kuka.IsGlobalPoint=False; Kuka.PointName=HP140; Kuka.BlendingEnabled=False; Kuka.MoveDataPtpName=PDAT35; Kuka.VelocityPtp=100; Kuka.CurrentCDSetIndex=0; Kuka.MovementParameterFieldEnabled=True; IlfCommand=PTP
;ENDFOLD
$BWDSTART = FALSE
PDAT_ACT = PPDAT35
FDAT_ACT = FHP140
BAS(#PTP_PARAMS, 100.0)
SET_CD_PARAMS (0)
PTP XHP140
;ENDFOLD
;FOLD PTP HP145 Vel=100 % PDAT36 Tool[64]:Zero Base[64]:Zero ;%{PE}
;FOLD Parameters ;%{h}
;Params IlfProvider=kukaroboter.basistech.inlineforms.movement.old; Kuka.IsGlobalPoint=False; Kuka.PointName=HP145; Kuka.BlendingEnabled=False; Kuka.MoveDataPtpName=PDAT36; Kuka.VelocityPtp=100; Kuka.CurrentCDSetIndex=0; Kuka.MovementParameterFieldEnabled=True; IlfCommand=PTP
;ENDFOLD
$BWDSTART = FALSE
PDAT_ACT = PPDAT36
FDAT_ACT = FHP145
BAS(#PTP_PARAMS, 100.0)
SET_CD_PARAMS (0)
PTP XHP145
;ENDFOLD

;*******************************
;fold Alle Kontrollspitzen entfernen
MSG_BTN("OK")
MSG_SHOW("DAI_H_PROG",#dialog,999,"dai_rob_ok_4",handle,answer)
;endfold
;FOLD WAIT FOR ( IN 1026 'Vordefinierte Eingang immer ruckgesetzt.' )  ;%{PE}
;FOLD Parameters ;%{h}
;Params IlfProvider=kukaroboter.basistech.inlineforms.logics.waitfor; Kuka.WaitLogicTerm1=None; Kuka.WaitForNot1=False; Kuka.WaitLogicOp2.Term1=None; Kuka.WaitForNot2.Term1=False; Kuka.WaitForSysVar2.Term1=IN; Kuka.WaitForIndex2.Term1=1026; Kuka.WaitForIndexName2.Term1=Vordefinierte Eingang immer ruckgesetzt.; Kuka.WaitForTermNumbers=1; Kuka.WaitForOpNumbers=2; Kuka.WaitForCont=False
;ENDFOLD
WAIT FOR  ( $IN[1026] )
;ENDFOLD

;*******************************
;FOLD PTP HOME Vel=100 % DEFAULT;%{PE}
;FOLD Parameters ;%{h}
;Params IlfProvider=kukaroboter.basistech.inlineforms.movement.old; Kuka.IsGlobalPoint=False; Kuka.PointName=HOME; Kuka.BlendingEnabled=False; Kuka.MoveDataPtpName=DEFAULT; Kuka.VelocityPtp=100; Kuka.CurrentCDSetIndex=0; Kuka.MovementParameterFieldEnabled=True; IlfCommand=PTP
;ENDFOLD
$BWDSTART = FALSE
PDAT_ACT = PDEFAULT
FDAT_ACT = FHOME
BAS(#PTP_PARAMS, 100.0)
SET_CD_PARAMS (0)
PTP XHOME
;ENDFOLD

END

--- DAI_CHECK_GRH_01.dat ---
&ACCESS RVO
&REL 40
&COMMENT Greiferpruefung
&PARAM TEMPLATE = C:\KRC\roboter\template\vg_appl
&PARAM DISKPATH = KRC:\R1\H_Prog
DEFDAT  DAI_CHECK_GRH_01
;FOLD EXTERNAL DECLARATIONS;%{PE}%MKUKATPBASIS,%CEXT,%VCOMMON,%P
;FOLD BASISTECH EXT;%{PE}%MKUKATPBASIS,%CEXT,%VEXT,%P
EXT  BAS (BAS_COMMAND  :IN,REAL  :IN )
DECL INT SUCCESS
;ENDFOLD (BASISTECH EXT)
;FOLD USER EXT;%{E}%MKUKATPUSER,%CEXT,%VEXT,%P
;Make your modifications here
;ENDFOLD (USER EXT)
;FOLD COLLISION
EXT  COLLSTOP (INT  :IN,INT  :IN )
;ENDFOLD  (Collision)
;ENDFOLD (EXTERNAL DECLERATIONS)
DECL INT handle,answer
DECL BASIS_SUGG_T LAST_BASIS={POINT1[] "P0                      ",POINT2[] "P0                      ",CP_PARAMS[] "CPDAT0                  ",PTP_PARAMS[] "PDAT0                   ",CONT[] "                        ",CP_VEL[] "2.0                     ",PTP_VEL[] "100                     ",SYNC_PARAMS[] "SYNCDAT                 ",SPL_NAME[] "S0                      ",A_PARAMS[] "ADAT0                   "}
DECL MODULEPARAM_T LAST_TP_PARAMS={PARAMS[] "Kuka.Content=Kontrollposition 6 QM2MM2 mit Tool 64; Kuka.PointName=CONTROL6; Kuka.FrameData.base_no=64; Kuka.FrameData.tool_no=64; Kuka.FrameData.ipo_frame=#BASE; Kuka.FrameData.point2=; Kuka.isglobalpoint=False; Kuka.MoveDataPtpName=PDAT44; Kuka.MovementDataPdat.apo_mode=#CDIS; Kuka.MovementDataPdat.apo_dist=0; Kuka.MovementData.vel=0.2; Kuka.MovementData.acc=100; Kuka.MovementData.exax_ign=0; Kuka.VelocityPtp=100; Kuka.BlendingEnabled=False; Kuka.APXEnabled=False; Kuka.CurrentCDSetIndex=0; Kuka.MoveDataName=CPDAT39; Kuka.MovementData.cb={AUX_PT {ORI #CONSIDER,E1 #CONSIDER,E2 #CONSIDER,E3 #CONSIDER,E4 #CONSIDER,E5 #CONSIDER,E6 #CONSIDER},TARGET_PT {ORI #INTERPOLATE,E1 #INTERPOLATE,E2 #INTERPOLATE,E3 #INTERPOLATE,E4 #INTERPOLATE,E5 #INTERPOLATE,E6 #INTERPOLATE}}; Kuka.MovementData.apo_fac=50; Kuka.MovementData.apo_dist=0; Kuka.MovementData.axis_acc=100; Kuka.MovementData.axis_vel=100; Kuka.MovementData.circ_typ=#BASE; Kuka.MovementData.jerk_fac=50; Kuka.MovementData.ori_typ=#VAR; Kuka.VelocityPath=0.2"}

; E6POS Declarations
DECL E6POS XHP005={X 2063.29907,Y 88.3752747,Z 2504.77905,A -96.9149857,B 34.1415215,C -134.511780,S 18,T 10,E1 -700.000,E2 0.0,E3 0.0,E4 0.0,E5 0.0,E6 0.0}
DECL E6POS XHP010={X 2266.63428,Y 1104.36121,Z 1217.34045,A 49.6174126,B 153.307922,C -29.7535686,S 18,T 11,E1 -700.000,E2 0.0,E3 0.0,E4 0.0,E5 0.0,E6 0.0}
DECL E6POS XHP015={X 2268.97266,Y 1112.12195,Z 943.869690,A -130.946686,B 16.1870270,C 144.242569,S 18,T 11,E1 -700.000,E2 0.0,E3 0.0,E4 0.0,E5 0.0,E6 0.0}
DECL E6POS XCONTROL1={X 2268.98633,Y 1112.12817,Z 893.224182,A -130.946945,B 16.1865253,C 144.241669,S 18,T 11,E1 -700.000,E2 0.0,E3 0.0,E4 0.0,E5 0.0,E6 0.0}
DECL E6POS XHP020={X 2268.97266,Y 1112.12195,Z 943.869690,A -130.946686,B 16.1870270,C 144.242569,S 18,T 11,E1 -700.000,E2 0.0,E3 0.0,E4 0.0,E5 0.0,E6 0.0}
DECL E6POS XHP025={X 2757.79614,Y 1451.10266,Z 514.305908,A -43.5338211,B -8.90570450,C -163.666183,S 18,T 11,E1 -700.000,E2 0.0,E3 0.0,E4 0.0,E5 0.0,E6 0.0}
DECL E6POS XCONTROL1A={X 2757.81250,Y 1451.10559,Z 463.700,A -43.5339928,B -8.90535545,C -163.665344,S 18,T 11,E1 -700.000,E2 0.0,E3 0.0,E4 0.0,E5 0.0,E6 0.0}
DECL E6POS XHP030={X 2757.79614,Y 1451.10266,Z 514.305908,A -43.5338211,B -8.90570450,C -163.666183,S 18,T 11,E1 -700.000,E2 0.0,E3 0.0,E4 0.0,E5 0.0,E6 0.0}
DECL E6POS XHP035={X 2356.66064,Y 1457.32861,Z 1332.30847,A -155.000259,B 0.00141960150,C 135.000336,S 18,T 11,E1 -700.000,E2 0.0,E3 0.0,E4 0.0,E5 0.0,E6 0.0}
DECL E6POS XCONTROL2={X 2356.72119,Y 1457.34119,Z 1174.66858,A -155.000076,B -9.80291952E-05,C 134.999817,S 18,T 11,E1 -700.000,E2 0.0,E3 0.0,E4 0.0,E5 0.0,E6 0.0}
DECL E6POS XHP040={X 2356.66064,Y 1457.32861,Z 1332.30847,A -155.000259,B 0.00141960150,C 135.000336,S 18,T 11,E1 -700.000,E2 0.0,E3 0.0,E4 0.0,E5 0.0,E6 0.0}
DECL E6POS XHP045={X 2319.93408,Y 1413.50757,Z 1808.81506,A 93.2296677,B 147.332504,C 1.51159179,S 18,T 11,E1 -700.000,E2 0.0,E3 0.0,E4 0.0,E5 0.0,E6 0.0}
DECL E6POS XHP050={X 2262.64893,Y 1283.55750,Z 1545.77563,A -20.0800247,B 8.71057510,C 158.799774,S 18,T 3,E1 -700.000,E2 0.0,E3 0.0,E4 0.0,E5 0.0,E6 0.0}
DECL E6POS XHP055={X 2383.32031,Y 1379.64563,Z 1144.32092,A -21.8058491,B 13.5951395,C 149.902588,S 18,T 3,E1 -700.000,E2 0.0,E3 0.0,E4 0.0,E5 0.0,E6 0.0}
DECL E6POS XCONTROL3={X 2383.33130,Y 1379.64734,Z 1112.70752,A -21.8059864,B 13.5954123,C 149.902588,S 18,T 3,E1 -700.000,E2 0.0,E3 0.0,E4 0.0,E5 0.0,E6 0.0}
DECL E6POS XHP060={X 2383.32031,Y 1379.64563,Z 1144.32092,A -21.8058491,B 13.5951395,C 149.902588,S 18,T 3,E1 -700.000,E2 0.0,E3 0.0,E4 0.0,E5 0.0,E6 0.0}
DECL E6POS XHP065={X 2361.85181,Y 1292.55591,Z 1248.06311,A -28.2764454,B 9.64973,C 147.561890,S 18,T 3,E1 -700.000,E2 0.0,E3 0.0,E4 0.0,E5 0.0,E6 0.0}
DECL E6POS XCONTROL4={X 2361.88,Y 1292.56079,Z 1175.28552,A -28.2766495,B 9.65033531,C 147.561829,S 18,T 3,E1 -700.000,E2 0.0,E3 0.0,E4 0.0,E5 0.0,E6 0.0}
DECL E6POS XHP070={X 2361.85181,Y 1292.55591,Z 1248.06311,A -28.2764454,B 9.64973,C 147.561890,S 18,T 3,E1 -700.000,E2 0.0,E3 0.0,E4 0.0,E5 0.0,E6 0.0}
DECL E6POS XHP075={X 2304.85913,Y 1252.16748,Z 1531.96204,A -27.0462933,B 5.61871767,C 156.797379,S 18,T 3,E1 -700.000,E2 0.0,E3 0.0,E4 0.0,E5 0.0,E6 0.0}
DECL E6POS XHP080={X 2293.75513,Y 1172.40491,Z 1558.79590,A 69.9164352,B 146.264679,C -5.13508368,S 18,T 11,E1 -700.000,E2 0.0,E3 0.0,E4 0.0,E5 0.0,E6 0.0}
DECL E6POS XHP085={X 2758.63281,Y 440.551086,Z 828.448364,A 35.6698914,B -176.662216,C -37.7142868,S 18,T 11,E1 -700.000,E2 0.0,E3 0.0,E4 0.0,E5 0.0,E6 0.0}
DECL E6POS XHP090={X 2805.59497,Y 436.801819,Z 639.113770,A -140.264801,B -4.52814770,C 139.532959,S 18,T 11,E1 -700.000,E2 0.0,E3 0.0,E4 0.0,E5 0.0,E6 0.0}
DECL E6POS XCONTROL5={X 2778.99536,Y 436.352570,Z 510.966522,A -140.265945,B -4.52816916,C 139.531570,S 18,T 11,E1 -700.000,E2 0.0,E3 0.0,E4 0.0,E5 0.0,E6 0.0}
DECL E6POS XHP095={X 2805.59497,Y 436.801819,Z 639.113770,A -140.264801,B -4.52814770,C 139.532959,S 18,T 11,E1 -700.000,E2 0.0,E3 0.0,E4 0.0,E5 0.0,E6 0.0}
DECL E6POS XHP100={X 2730.29541,Y 443.548676,Z 1127.03931,A -140.588135,B 0.526392102,C 140.706696,S 18,T 11,E1 -700.000,E2 0.0,E3 0.0,E4 0.0,E5 0.0,E6 0.0}
DECL E6POS XHP105={X 2181.47852,Y 393.179901,Z 2034.91248,A -138.476685,B 40.7378464,C 170.675598,S 18,T 11,E1 -400.000,E2 0.0,E3 0.0,E4 0.0,E5 0.0,E6 0.0}
DECL E6POS XHP110={X 1986.98828,Y 455.080292,Z 1735.26514,A -73.6478729,B -22.4779110,C -132.601166,S 18,T 3,E1 -400.000,E2 0.0,E3 0.0,E4 0.0,E5 0.0,E6 0.0}
DECL E6POS XHP115={X 1763.97400,Y 585.713806,Z 1418.68872,A 37.2463837,B -48.7374115,C 148.730087,S 18,T 3,E1 -400.000,E2 0.0,E3 0.0,E4 0.0,E5 0.0,E6 0.0}
DECL E6POS XHP120={X 1744.35962,Y 805.534302,Z 999.566650,A 84.2576141,B -14.0044260,C 147.188278,S 18,T 3,E1 -400.000,E2 0.0,E3 0.0,E4 0.0,E5 0.0,E6 0.0}
DECL E6POS XHP125={X 1915.26221,Y 864.236511,Z 669.903259,A 82.7754,B -7.65904474,C 155.059280,S 18,T 3,E1 -400.000,E2 0.0,E3 0.0,E4 0.0,E5 0.0,E6 0.0}
DECL E6POS XCONTROL6={X 1915.25903,Y 864.251770,Z 580.404419,A 82.7733917,B -7.65879822,C 155.062271,S 18,T 3,E1 -400.000,E2 0.0,E3 0.0,E4 0.0,E5 0.0,E6 0.0}
DECL E6POS XHP130={X 1915.26221,Y 864.236511,Z 669.903259,A 82.7754,B -7.65904474,C 155.059280,S 18,T 3,E1 -400.000,E2 0.0,E3 0.0,E4 0.0,E5 0.0,E6 0.0}
DECL E6POS XHP135={X 1744.36084,Y 805.535,Z 999.561523,A 84.2576065,B -14.0044270,C 147.188293,S 18,T 3,E1 -400.000,E2 0.0,E3 0.0,E4 0.0,E5 0.0,E6 0.0}
DECL E6POS XHP140={X 1523.88611,Y 520.430,Z 1649.99036,A 23.3499794,B -61.8450661,C 150.255859,S 18,T 3,E1 -400.000,E2 0.0,E3 0.0,E4 0.0,E5 0.0,E6 0.0}
DECL E6POS XHP145={X 1662.63062,Y 151.029282,Z 2290.65259,A -86.4169617,B -34.0953102,C -120.930328,S 18,T 3,E1 -460.888611,E2 0.0,E3 0.0,E4 0.0,E5 0.0,E6 0.0}

; PDAT/LDAT Declarations
DECL PDAT PPDAT1={VEL 100.000,ACC 100.000,APO_DIST 0.0,APO_MODE #CDIS,GEAR_JERK 50.0000,EXAX_IGN 0}
DECL PDAT PPDAT2={VEL 100.000,ACC 100.000,APO_DIST 0.0,APO_MODE #CDIS,GEAR_JERK 50.0000,EXAX_IGN 0}
DECL PDAT PPDAT3={VEL 100.000,ACC 100.000,APO_DIST 0.0,APO_MODE #CDIS,GEAR_JERK 50.0000,EXAX_IGN 0}
DECL LDAT LCPDAT4={VEL 0.200000,ACC 100.000,APO_DIST 0.0,APO_FAC 50.0000,AXIS_VEL 100.000,AXIS_ACC 100.000,ORI_TYP #VAR,CIRC_TYP #BASE,JERK_FAC 50.0000,GEAR_JERK 50.0000,EXAX_IGN 0}
DECL LDAT LCPDAT5={VEL 0.200000,ACC 100.000,APO_DIST 0.0,APO_FAC 50.0000,AXIS_VEL 100.000,AXIS_ACC 100.000,ORI_TYP #VAR,CIRC_TYP #BASE,JERK_FAC 50.0000,GEAR_JERK 50.0000,EXAX_IGN 0}
DECL PDAT PPDAT6={VEL 100.000,ACC 100.000,APO_DIST 0.0,APO_MODE #CDIS,GEAR_JERK 50.0000,EXAX_IGN 0}
DECL LDAT LCPDAT7={VEL 0.200000,ACC 100.000,APO_DIST 0.0,APO_FAC 50.0000,AXIS_VEL 100.000,AXIS_ACC 100.000,ORI_TYP #VAR,CIRC_TYP #BASE,JERK_FAC 50.0000,GEAR_JERK 50.0000,EXAX_IGN 0}
DECL LDAT LCPDAT8={VEL 0.200000,ACC 100.000,APO_DIST 0.0,APO_FAC 50.0000,AXIS_VEL 100.000,AXIS_ACC 100.000,ORI_TYP #VAR,CIRC_TYP #BASE,JERK_FAC 50.0000,GEAR_JERK 50.0000,EXAX_IGN 0}
DECL PDAT PPDAT9={VEL 100.000,ACC 100.000,APO_DIST 0.0,APO_MODE #CDIS,GEAR_JERK 50.0000,EXAX_IGN 0}
DECL LDAT LCPDAT10={VEL 0.200000,ACC 100.000,APO_DIST 0.0,APO_FAC 50.0000,AXIS_VEL 100.000,AXIS_ACC 100.000,ORI_TYP #VAR,CIRC_TYP #BASE,JERK_FAC 50.0000,GEAR_JERK 50.0000,EXAX_IGN 0}
DECL LDAT LCPDAT11={VEL 0.200000,ACC 100.000,APO_DIST 0.0,APO_FAC 50.0000,AXIS_VEL 100.000,AXIS_ACC 100.000,ORI_TYP #VAR,CIRC_TYP #BASE,JERK_FAC 50.0000,GEAR_JERK 50.0000,EXAX_IGN 0}
DECL PDAT PPDAT12={VEL 100.000,ACC 100.000,APO_DIST 0.0,APO_MODE #CDIS,GEAR_JERK 50.0000,EXAX_IGN 0}
DECL PDAT PPDAT13={VEL 100.000,ACC 100.000,APO_DIST 0.0,APO_MODE #CDIS,GEAR_JERK 50.0000,EXAX_IGN 0}
DECL PDAT PPDAT14={VEL 100.000,ACC 100.000,APO_DIST 0.0,APO_MODE #CDIS,GEAR_JERK 50.0000,EXAX_IGN 0}
DECL LDAT LCPDAT15={VEL 0.200000,ACC 100.000,APO_DIST 0.0,APO_FAC 50.0000,AXIS_VEL 100.000,AXIS_ACC 100.000,ORI_TYP #VAR,CIRC_TYP #BASE,JERK_FAC 50.0000,GEAR_JERK 50.0000,EXAX_IGN 0}
DECL LDAT LCPDAT16={VEL 0.200000,ACC 100.000,APO_DIST 0.0,APO_FAC 50.0000,AXIS_VEL 100.000,AXIS_ACC 100.000,ORI_TYP #VAR,CIRC_TYP #BASE,JERK_FAC 50.0000,GEAR_JERK 50.0000,EXAX_IGN 0}
DECL PDAT PPDAT17={VEL 100.000,ACC 100.000,APO_DIST 0.0,APO_MODE #CDIS,GEAR_JERK 50.0000,EXAX_IGN 0}
DECL LDAT LCPDAT18={VEL 0.200000,ACC 100.000,APO_DIST 0.0,APO_FAC 50.0000,AXIS_VEL 100.000,AXIS_ACC 100.000,ORI_TYP #VAR,CIRC_TYP #BASE,JERK_FAC 50.0000,GEAR_JERK 50.0000,EXAX_IGN 0}
DECL LDAT LCPDAT19={VEL 0.200000,ACC 100.000,APO_DIST 0.0,APO_FAC 50.0000,AXIS_VEL 100.000,AXIS_ACC 100.000,ORI_TYP #VAR,CIRC_TYP #BASE,JERK_FAC 50.0000,GEAR_JERK 50.0000,EXAX_IGN 0}
DECL PDAT PPDAT20={VEL 100.000,ACC 100.000,APO_DIST 0.0,APO_MODE #CDIS,GEAR_JERK 50.0000,EXAX_IGN 0}
DECL PDAT PPDAT21={VEL 100.000,ACC 100.000,APO_DIST 0.0,APO_MODE #CDIS,GEAR_JERK 50.0000,EXAX_IGN 0}
DECL PDAT PPDAT22={VEL 100.000,ACC 100.000,APO_DIST 0.0,APO_MODE #CDIS,GEAR_JERK 50.0000,EXAX_IGN 0}
DECL PDAT PPDAT23={VEL 100.000,ACC 100.000,APO_DIST 0.0,APO_MODE #CDIS,GEAR_JERK 50.0000,EXAX_IGN 0}
DECL LDAT LCPDAT24={VEL 0.200000,ACC 100.000,APO_DIST 0.0,APO_FAC 50.0000,AXIS_VEL 100.000,AXIS_ACC 100.000,ORI_TYP #VAR,CIRC_TYP #BASE,JERK_FAC 50.0000,GEAR_JERK 50.0000,EXAX_IGN 0}
DECL LDAT LCPDAT25={VEL 0.200000,ACC 100.000,APO_DIST 0.0,APO_FAC 50.0000,AXIS_VEL 100.000,AXIS_ACC 100.000,ORI_TYP #VAR,CIRC_TYP #BASE,JERK_FAC 50.0000,GEAR_JERK 50.0000,EXAX_IGN 0}
DECL PDAT PPDAT26={VEL 100.000,ACC 100.000,APO_DIST 0.0,APO_MODE #CDIS,GEAR_JERK 50.0000,EXAX_IGN 0}
DECL PDAT PPDAT27={VEL 100.000,ACC 100.000,APO_DIST 0.0,APO_MODE #CDIS,GEAR_JERK 50.0000,EXAX_IGN 0}
DECL PDAT PPDAT28={VEL 100.000,ACC 100.000,APO_DIST 0.0,APO_MODE #CDIS,GEAR_JERK 50.0000,EXAX_IGN 0}
DECL PDAT PPDAT29={VEL 100.000,ACC 100.000,APO_DIST 0.0,APO_MODE #CDIS,GEAR_JERK 50.0000,EXAX_IGN 0}
DECL PDAT PPDAT30={VEL 100.000,ACC 100.000,APO_DIST 0.0,APO_MODE #CDIS,GEAR_JERK 50.0000,EXAX_IGN 0}
DECL PDAT PPDAT31={VEL 100.000,ACC 100.000,APO_DIST 0.0,APO_MODE #CDIS,GEAR_JERK 50.0000,EXAX_IGN 0}
DECL LDAT LCPDAT32={VEL 0.200000,ACC 100.000,APO_DIST 0.0,APO_FAC 50.0000,AXIS_VEL 100.000,AXIS_ACC 100.000,ORI_TYP #VAR,CIRC_TYP #BASE,JERK_FAC 50.0000,GEAR_JERK 50.0000,EXAX_IGN 0,CB {AUX_PT {ORI #CONSIDER,E1 #CONSIDER,E2 #CONSIDER,E3 #CONSIDER,E4 #CONSIDER,E5 #CONSIDER,E6 #CONSIDER},TARGET_PT {ORI #INTERPOLATE,E1 #INTERPOLATE,E2 #INTERPOLATE,E3 #INTERPOLATE,E4 #INTERPOLATE,E5 #INTERPOLATE,E6 #INTERPOLATE}}}
DECL LDAT LCPDAT33={VEL 0.200000,ACC 100.000,APO_DIST 0.0,APO_FAC 50.0000,AXIS_VEL 100.000,AXIS_ACC 100.000,ORI_TYP #VAR,CIRC_TYP #BASE,JERK_FAC 50.0000,GEAR_JERK 50.0000,EXAX_IGN 0}
DECL PDAT PPDAT34={VEL 100.000,ACC 100.000,APO_DIST 0.0,APO_MODE #CDIS,GEAR_JERK 50.0000,EXAX_IGN 0}
DECL PDAT PPDAT35={VEL 100.000,ACC 100.000,APO_DIST 0.0,APO_MODE #CDIS,GEAR_JERK 50.0000,EXAX_IGN 0}
DECL PDAT PPDAT36={VEL 100.000,ACC 100.000,APO_DIST 0.0,APO_MODE #CDIS,GEAR_JERK 50.0000,EXAX_IGN 0}

; FDAT Declarations
DECL FDAT FHOME={TOOL_NO 64,BASE_NO 64,IPO_FRAME #BASE,POINT2[] " "}
DECL FDAT FHP005={TOOL_NO 64,BASE_NO 64,IPO_FRAME #BASE,POINT2[] " "}
DECL FDAT FHP010={TOOL_NO 64,BASE_NO 64,IPO_FRAME #BASE,POINT2[] " "}
DECL FDAT FHP015={TOOL_NO 64,BASE_NO 64,IPO_FRAME #BASE,POINT2[] " "}
DECL FDAT FCONTROL1={TOOL_NO 64,BASE_NO 64,IPO_FRAME #BASE,POINT2[] " "}
DECL FDAT FHP020={TOOL_NO 64,BASE_NO 64,IPO_FRAME #BASE,POINT2[] " "}
DECL FDAT FHP025={TOOL_NO 10,BASE_NO 64,IPO_FRAME #BASE,POINT2[] " "}
DECL FDAT FCONTROL1A={TOOL_NO 10,BASE_NO 64,IPO_FRAME #BASE,POINT2[] " "}
DECL FDAT FHP030={TOOL_NO 10,BASE_NO 64,IPO_FRAME #BASE,POINT2[] " "}
DECL FDAT FHP035={TOOL_NO 64,BASE_NO 64,IPO_FRAME #BASE,POINT2[] " "}
DECL FDAT FCONTROL2={TOOL_NO 64,BASE_NO 64,IPO_FRAME #BASE,POINT2[] " "}
DECL FDAT FHP040={TOOL_NO 64,BASE_NO 64,IPO_FRAME #BASE,POINT2[] " "}
DECL FDAT FHP045={TOOL_NO 64,BASE_NO 64,IPO_FRAME #BASE,POINT2[] " "}
DECL FDAT FHP050={TOOL_NO 64,BASE_NO 64,IPO_FRAME #BASE,POINT2[] " "}
DECL FDAT FHP055={TOOL_NO 64,BASE_NO 64,IPO_FRAME #BASE,POINT2[] " "}
DECL FDAT FCONTROL3={TOOL_NO 64,BASE_NO 64,IPO_FRAME #BASE,POINT2[] " "}
DECL FDAT FHP060={TOOL_NO 64,BASE_NO 64,IPO_FRAME #BASE,POINT2[] " "}
DECL FDAT FHP065={TOOL_NO 64,BASE_NO 64,IPO_FRAME #BASE,POINT2[] " "}
DECL FDAT FCONTROL4={TOOL_NO 64,BASE_NO 64,IPO_FRAME #BASE,POINT2[] " "}
DECL FDAT FHP070={TOOL_NO 64,BASE_NO 64,IPO_FRAME #BASE,POINT2[] " "}
DECL FDAT FHP075={TOOL_NO 64,BASE_NO 64,IPO_FRAME #BASE,POINT2[] " "}
DECL FDAT FHP080={TOOL_NO 64,BASE_NO 64,IPO_FRAME #BASE,POINT2[] " "}
DECL FDAT FHP085={TOOL_NO 64,BASE_NO 64,IPO_FRAME #BASE,POINT2[] " "}
DECL FDAT FHP090={TOOL_NO 64,BASE_NO 64,IPO_FRAME #BASE,POINT2[] " "}
DECL FDAT FCONTROL5={TOOL_NO 64,BASE_NO 64,IPO_FRAME #BASE,POINT2[] " "}
DECL FDAT FHP095={TOOL_NO 64,BASE_NO 64,IPO_FRAME #BASE,POINT2[] " "}
DECL FDAT FHP100={TOOL_NO 64,BASE_NO 64,IPO_FRAME #BASE,POINT2[] " "}
DECL FDAT FHP105={TOOL_NO 64,BASE_NO 64,IPO_FRAME #BASE,POINT2[] " "}
DECL FDAT FHP110={TOOL_NO 64,BASE_NO 64,IPO_FRAME #BASE,POINT2[] " "}
DECL FDAT FHP115={TOOL_NO 64,BASE_NO 64,IPO_FRAME #BASE,POINT2[] " "}
DECL FDAT FHP120={TOOL_NO 64,BASE_NO 64,IPO_FRAME #BASE,POINT2[] " "}
DECL FDAT FHP125={TOOL_NO 64,BASE_NO 64,IPO_FRAME #BASE,POINT2[] " "}
DECL FDAT FCONTROL6={TOOL_NO 64,BASE_NO 64,IPO_FRAME #BASE,POINT2[] " "}
DECL FDAT FHP130={TOOL_NO 64,BASE_NO 64,IPO_FRAME #BASE,POINT2[] " "}
DECL FDAT FHP135={TOOL_NO 64,BASE_NO 64,IPO_FRAME #BASE,POINT2[] " "}
DECL FDAT FHP140={TOOL_NO 64,BASE_NO 64,IPO_FRAME #BASE,POINT2[] " "}
DECL FDAT FHP145={TOOL_NO 64,BASE_NO 64,IPO_FRAME #BASE,POINT2[] " "}

ENDDAT
